FUNCTION_BLOCK lichten
VAR_INPUT
	Toggle 	: BOOL;
	ON 		: BOOL;
	OFF		: BOOL;
	Enable 	: BOOL;
END_VAR
VAR_OUTPUT
	lamp 	: BOOL;
	Q		: BOOL;	// puls 100ms
END_VAR
VAR
	pLamp	: BOOL;
	pToggle : BOOL;
	pON 	: BOOL;
	pOFF	: BOOL;
	puls	: TP;
END_VAR

pLamp := lamp;

IF Toggle THEN pToggle := TRUE; END_IF
IF ON THEN pON := TRUE; END_IF
IF OFF THEN pOFF := TRUE; END_IF

IF Enable AND NOT(puls.Q) THEN
	IF pON THEN lamp := TRUE; pON := FALSE;
	ELSIF pOFF THEN lamp := FALSE; pOFF := FALSE;
	ELSIF pToggle THEN lamp := NOT lamp; pToggle := FALSE;
	END_IF;
END_IF

IF lamp <> pLamp THEN puls.IN := TRUE; ELSE puls.IN := FALSE; END_IF

puls(PT := T#250MS, Q => Q);

END_FUNCTION_BLOCK

(* stored: Version 1.1.0.1, ProductVersion 3.1.4022.12
   POU lichten: Id {11dffa0e-0bd9-4182-a8c0-07e0ca83ba60}, SpecialFunc None *)
